PROGRAM Pneumatics_Template
VAR
END_VAR

//Test the program to control pneumatic acutator through PneumaticsVisu.
//Currently implemented control of single solenoid through PLC and and manually, with two momentary push buttons.

END_PROGRAM

(* stored: Version 1.1.0.1, ProductVersion 3.1.4024.12
   POU Pneumatics_Template: Id {7bf401fb-a600-4741-a67b-36f20e194cfc}, SpecialFunc None *)
